# EPICS autosave request: iocBoot/sioc-b084-im02/sioc-b084-im02.req
file "facet2.req" AREA=IN10,POS=791
